{attribute addProperty BoxType "EK1322-0000-0017"}
{attribute addProperty Id "Status_UsAT %I*Status_Us_D944C060810Status_UpAT %I*Status_Up_D944C060810WcStateAT %I*WcState_98A4DF7520.250InfoDataAT %I*InfoData_192954DE1620"}
{attribute addProperty CRC "793642750"}
{attribute addProperty SizeInBites "34"}
{attribute addProperty SizeInBytes "4.25"}
TYPE EK1322_0EEAC8F2 :
STRUCT
	{attribute addProperty Name "Status_Us"}
	Status_Us : Status_Us_D944C060;
	{attribute addProperty Name "Status_Up"}
	Status_Up : Status_Up_D944C060;
	{attribute addProperty Name "WcState"}
	WcState : WcState_98A4DF75;
	{attribute addProperty Name "InfoData"}
	InfoData : InfoData_192954DE;
END_STRUCT
END_TYPE

(* stored: Version 1.2.0.0, ProductVersion 3.1.4024.9
   DUT EK1322_0EEAC8F2: Id {e8b8e3b6-ae55-40b7-87a1-57f01f028e41} *)
